TYPE ResponseData : 
STRUCT
	Header : STRING(Constants.HEADER_STRING_SIZE);
	Payload : STRING(Constants.PAYLOAD_STRING_SIZE);
END_STRUCT
END_TYPE

(* stored: Version 1.1.0.1, ProductVersion 3.1.4024.12
   DUT ResponseData: Id {4e17831c-a1b5-0bef-3931-0a7033ba3813} *)
